// TIA Portal V19 export
VAR_GLOBAL   // PLC tag table "Default tag table"
   "Conveyor 0" AT %Q0.0 : Bool;
   "memory-eme" AT %M0.0 : Bool;
END_VAR
